ABB RAPID module: Wizard.modx

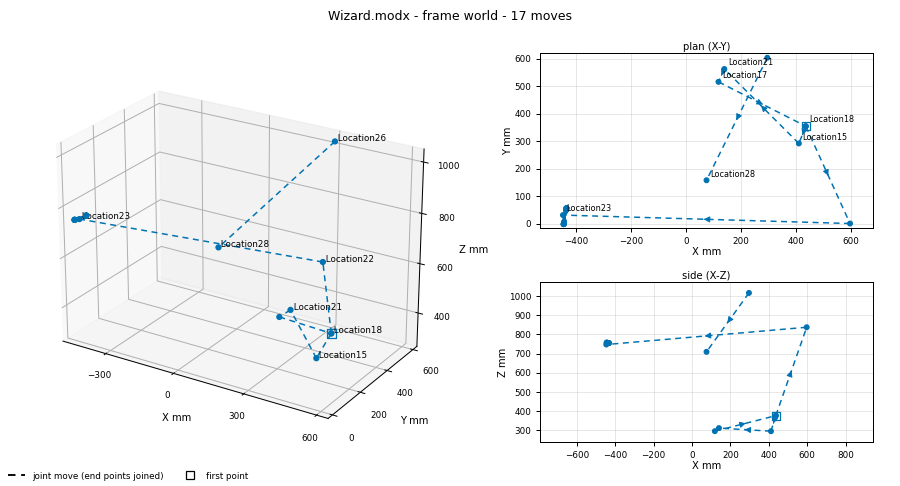
[picture p0: tool path of Wizard.modx in frame world, 17 of 19 moves have a stored position in this frame; points joined in program order, loops and branches not executed]
MODULE Wizard
PERS robtarget Location1:=[[141.020217895508, 436.321899414063, 575.21875], [0.017813965678215, 0.999827980995178, -0.000279141531791538, -0.0051563223823905], [0, -1, -2, 0], [9000000000, 9000000000, 9000000000, 9000000000, 9000000000, 9000000000]];
PERS robtarget Location2:=[[508.657287597656, 345.39111328125, 565.002990722656], [0.027114637196064, 0.945273578166962, -0.324619859457016, -0.018564136698842], [0, -1, -2, 0], [9000000000, 9000000000, 9000000000, 9000000000, 9000000000, 9000000000]];
PERS robtarget Location3:=[[138.697784423828, 217.932708740234, 413.045196533203], [0.07676836848259, 0.98807281255722, -0.127942427992821, -0.038071520626545], [0, 0, -2, 0], [9000000000, 9000000000, 9000000000, 9000000000, 9000000000, 9000000000]];
PERS robtarget Location4:=[[-51.5362167358398, 430.496246337891, 337.229919433594], [0.0170931983739138, -0.979323327541351, -0.201356798410416, 0.0094364807009697], [1, 0, -2, 0], [9000000000, 9000000000, 9000000000, 9000000000, 9000000000, 9000000000]];
PERS robtarget Location5:=[[-45.3218955993652, 414.107299804688, 542.560546875], [0.0331718660891056, 0.974595308303833, 0.220419079065323, 0.0218859035521746], [1, -1, -2, 0], [9000000000, 9000000000, 9000000000, 9000000000, 9000000000, 9000000000]];
PERS robtarget Location6:=[[-42.930736541748, 416.871459960938, 368.191131591797], [0.0221891868859529, 0.973919808864594, 0.225001737475395, 0.0190272349864244], [1, -1, -2, 0], [9000000000, 9000000000, 9000000000, 9000000000, 9000000000, 9000000000]];
PERS robtarget Location7:=[[-34.9866142272949, 458.268798828125, 584.186340332031], [0.00795904919505119, -0.978147804737091, -0.205494686961174, -0.0305846277624369], [1, -1, -2, 0], [9000000000, 9000000000, 9000000000, 9000000000, 9000000000, 9000000000]];
PERS robtarget Location8:=[[145.745910644531, 420.857421875, 492.48779296875], [0.0239510629326105, -0.999478936195374, 0.0202637929469347, 0.00758857233449817], [0, 0, -2, 0], [9000000000, 9000000000, 9000000000, 9000000000, 9000000000, 9000000000]];
PERS robtarget Location9:=[[-560.7, 509.56, 592.15], [0.00123678, -0.378767, 0.925393, 0.0135282], [1, -1, 1, 0], [9000000000, 9000000000, 9000000000, 9000000000, 9000000000, 9000000000]];
PERS robtarget Location10:=[[613.03, 509.55, 592.16], [0.00125397, -0.378757, 0.925396, 0.0135404], [0, 0, -1, 0], [9000000000, 9000000000, 9000000000, 9000000000, 9000000000, 9000000000]];
PERS robtarget Location11:=[[60.7467308044434, 465.576812744141, 491.8779296875], [0.00205219932831824, -0.387099027633667, 0.921912610530853, 0.0150760682299733], [0, 0, 0, 0], [9000000000, 9000000000, 9000000000, 9000000000, 9000000000, 9000000000]];
PERS robtarget Location12:=[[60.7467498779297, 465.576934814453, 491.878173828125], [0.00205230480059981, -0.387099027633667, 0.921912610530853, 0.0150762461125851], [0, 0, 0, 0], [9000000000, 9000000000, 9000000000, 9000000000, 9000000000, 9000000000]];
PERS robtarget Location13:=[[41.1625862121582, 462.905975341797, 470.445495605469], [0.00223985756747425, -0.386858403682709, 0.922010123729706, 0.0152596672996879], [0, 0, 0, 0], [9000000000, 9000000000, 9000000000, 9000000000, 9000000000, 9000000000]];
PERS robtarget Location14:=[[351.474975585938, 309.715148925781, 260.885223388672], [0.0170289911329746, 0.976639628410339, -0.207100242376328, 0.0547224693000317], [0, -1, -2, 0], [9000000000, 9000000000, 9000000000, 9000000000, 9000000000, 9000000000]];
PERS robtarget Location15:=[[411.344787597656, 291.304351806641, 296.075225830078], [0.0101514291018248, 0.952983915805817, -0.300747394561768, 0.0356313996016979], [0, -1, -2, 0], [9000000000, 9000000000, 9000000000, 9000000000, 9000000000, 9000000000]];
PERS robtarget Location16:=[[411.403198242188, 291.338073730469, 296.152160644531], [0.010098023340106, 0.952989459037781, -0.300723135471344, 0.035703431814909], [0, -1, -2, 0], [9000000000, 9000000000, 9000000000, 9000000000, 9000000000, 9000000000]];
PERS robtarget Location17:=[[118.899482727051, 515.328552246094, 296.214111328125], [0.0189743582159281, -0.999544084072113, 0.0166813433170319, 0.0165309309959412], [0, 0, -2, 0], [9000000000, 9000000000, 9000000000, 9000000000, 9000000000, 9000000000]];
PERS robtarget Location18:=[[436.534332275391, 354.010101318359, 377.196624755859], [0.0128294415771961, -0.945383727550507, 0.325654596090317, 0.00584001466631889], [0, 0, -2, 0], [9000000000, 9000000000, 9000000000, 9000000000, 9000000000, 9000000000]];
PERS robtarget Location19:=[[155.497650146484, 559.769897460938, 283.121704101563], [0.0144326165318489, -0.999774158000946, 0.0155905513092875, -0.00053736986592412], [0, 0, -2, 0], [9000000000, 9000000000, 9000000000, 9000000000, 9000000000, 9000000000]];
PERS robtarget Location20:=[[156.645233154297, 546.048583984375, 292.123291015625], [0.0307666454464197, 0.998924672603607, -0.0285003632307053, -0.0197639297693968], [0, 0, -2, 0], [9000000000, 9000000000, 9000000000, 9000000000, 9000000000, 9000000000]];
PERS robtarget Location21:=[[140.207885742188, 562.077514648438, 312.297576904297], [0.0388302467763424, -0.999223053455353, 0.002286063041538, -0.00634820805862546], [0, 0, -2, 0], [9000000000, 9000000000, 9000000000, 9000000000, 9000000000, 9000000000]];
PERS robtarget Location22:=[[597.477416992188, -0.000894433644134551, 837.765869140625], [0.499986261129379, 8.83667325979332e-7, 0.866033315658569, 4.93338916385255e-7], [-1, 0, -1, 0], [9000000000, 9000000000, 9000000000, 9000000000, 9000000000, 9000000000]];
PERS robtarget Location23:=[[-446.701171875, 30.7164821624756, 747.700256347656], [0.00395846599712968, -0.956965982913971, -0.289376705884933, 0.0214827340096235], [1, 0, -1, 0], [9000000000, 9000000000, 9000000000, 9000000000, 9000000000, 9000000000]];
PERS robtarget Location24:=[[-444.170989990234, -2.30431890487671, 757.240234375], [0.144577205181122, 0.940973162651062, 0.294827669858932, -0.082119390368462], [1, 0, -1, 0], [9000000000, 9000000000, 9000000000, 9000000000, 9000000000, 9000000000]];
PERS robtarget Location25:=[[-434.068908691406, 55.5364799499512, 755.404907226563], [0.121449619531631, -0.952281355857849, -0.279508829116821, -0.0168841276317835], [1, -1, -1, 0], [9000000000, 9000000000, 9000000000, 9000000000, 9000000000, 9000000000]];
PERS robtarget Location26:=[[296.540557861328, 603.139465332031, 1016.55950927734], [0.525297164916992, -0.694388151168823, 0.491694390773773, 0.011160995811224], [0, -1, -1, 0], [9000000000, 9000000000, 9000000000, 9000000000, 9000000000, 9000000000]];
PERS robtarget Location27:=[[152.305084228516, 500.900573730469, 1112.82275390625], [0.541991829872131, -0.715796172618866, 0.435782372951508, 0.063042767345905], [0, -1, -1, 0], [9000000000, 9000000000, 9000000000, 9000000000, 9000000000, 9000000000]];
PERS robtarget Location28:=[[75.4926910400391, 157.420791625977, 709.636413574219], [0.00222255499102175, -0.525019109249115, -0.61897999048233, 0.584134995937347], [-2, -1, -1, 4], [9000000000, 9000000000, 9000000000, 9000000000, 9000000000, 9000000000]];
	PROC main()
MoveJ wi_homePosition, v1000, fine, tool0;
SetDO ABB_Local_IO_0_DO1, 1;
SetDO ABB_Local_IO_0_DO2, 0;
MoveJ Location18, v1000, fine, tool0;
MoveJ Location15, v1000, fine, tool0;
SetDO ABB_Local_IO_0_DO1, 0;
SetDO ABB_Local_IO_0_DO2, 1;
MoveJ Location21, v1000, fine, tool0;
MoveJ Location17, v1000, fine, tool0;
SetDO ABB_Local_IO_0_DO1, 1;
SetDO ABB_Local_IO_0_DO2, 0;
MoveJ Location18, v1000, fine, tool0;
SetDO ABB_Local_IO_0_DO1, 0;
SetDO ABB_Local_IO_0_DO2, 1;
MoveJ Location22, v1000, fine, tool0;
MoveJ Location23, v1000, fine, tool0;
SetDO ABB_Local_IO_0_DO1, 1;
SetDO ABB_Local_IO_0_DO2, 0;
MoveJ Location24, v1000, fine, tool0;
MoveJ Location25, v1000, fine, tool0;
SetDO ABB_Local_IO_0_DO1, 0;
SetDO ABB_Local_IO_0_DO2, 1;
SetDO ABB_Local_IO_0_DO1, 0;
SetDO ABB_Local_IO_0_DO2, 1;
MoveJ Location24, v1000, fine, tool0;
MoveJ Location25, v1000, fine, tool0;
MoveJ Location24, v1000, fine, tool0;
MoveJ Location25, v1000, fine, tool0;
MoveJ Location24, v1000, fine, tool0;
MoveJ Location25, v1000, fine, tool0;
MoveJ wi_homePosition, v1000, fine, tool0;
MoveJ Location26, v1000, fine, tool0;
MoveJ Location28, v1000, fine, tool0;
	ENDPROC
ENDMODULE
